FUNCTION_BLOCK FB_PID
VAR_INPUT
	i_bEnablePID		:BOOL	:=FALSE;
	i_rSetpoint			:REAL;				//required input from PLC logic
	i_rActual			:REAL;				//required input from PLC logic
	i_rKp				:REAL;
	i_rKi				:REAL;
	i_rKd				:REAL;
	i_rTdamp			:REAL;
	i_rOutMin			:REAL	:=0;
	i_rOutMax			:REAL	:=100;
	i_rManualOutput		:REAL	:=0;
	i_bEnablePWM		:BOOL	:=FALSE;
	i_iFreqPWM			:INT	:=1000;		//required input from PLC logic
	i_bAutotuneStart	:BOOL	:=FALSE;
	i_rAutotuneSetpoint	:REAL	:=0;
	i_bEnableAlarms		:BOOL;
	i_iHighAlarm		:INT;
	i_iHighWarning		:INT;
	i_iLowWarning		:INT;
	i_iLowAlarm			:INT;
	i_iWarningDelay		:INT;
	i_iAlarmDelay		:INT;
END_VAR
VAR_OUTPUT
	q_rOutputPID		:REAL;				//output for proportional control
	q_bOutputPWM		:BOOL;				//output for on/off control
	q_Difference		:REAL;
	q_AutotuneActive	:BOOL;
	q_AutotuneDone		:BOOL;
	i_sAutotuneTime		:STRING	:='00:00:00';
	q_rAutotuneKp		:REAL	:=0;
	q_rAutotuneKi		:REAL	:=0;
	q_rAutotuneKd		:REAL	:=0;
	q_bError			:BOOL;
	q_bErrorID			:INT	:=0;;
	q_bAlarmHigh		:BOOL;				
	q_bWarningHigh		:BOOL;
	q_bWarningLow		:BOOL;
	q_bAlarmLow			:BOOL;
END_VAR
VAR
	PID_AutoTuner		:FB_PID_AutoTuner;
	PWM_Autotune		:FB_PID_PWM;
	PID_Gain2Time		:FB_PID_Gain2Time;
	ST_PID_Params		:ST_CTRL_PID_PARAMS;
	PID_Control			:FB_CTRL_PID;
	PWM_Control			:FB_PID_PWM;
	M_Active_0			:FB_CTRL_PID;
	
	tonAlarmHigh		:TON;
	tonWarningHigh		:TON;
	tonWarningLow		:TON;
	tonAlarmLow			:TON;
	tonAutotuneTime		:TON;
	
END_VAR
VAR // added by the converter: edge detectors and wires of the graphical bodies
    _w1, _w2, _w3, _w4, _w5 : BOOL;
END_VAR

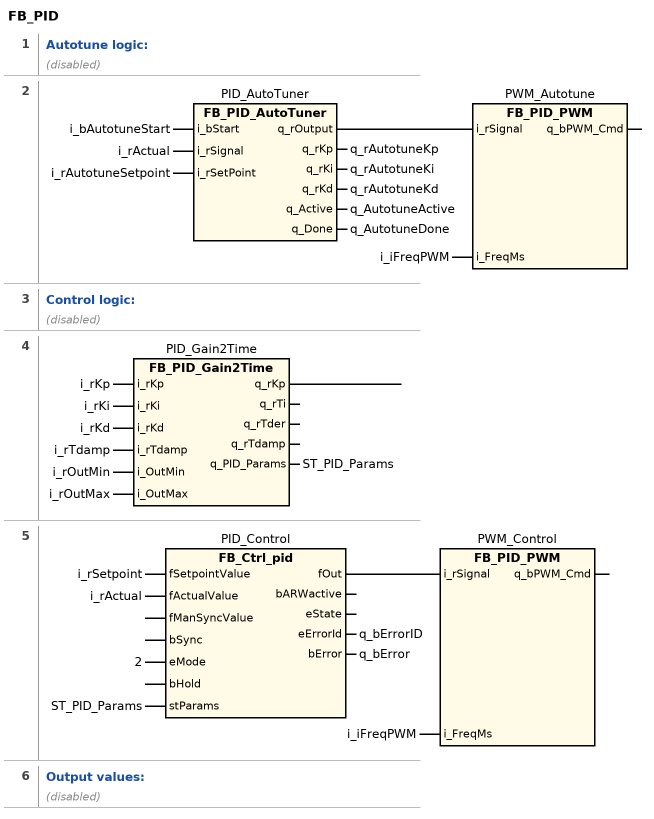
// NETWORK 1 (disabled)
// label: Autotune logic

// NETWORK 2
PID_AutoTuner(
    i_bStart := i_bAutotuneStart,
    i_rSignal := i_rActual,
    i_rSetPoint := i_rAutotuneSetpoint,
    q_rKp => q_rAutotuneKp,
    q_rKi => q_rAutotuneKi,
    q_rKd => q_rAutotuneKd,
    q_Active => q_AutotuneActive,
    q_Done => q_AutotuneDone); // FB_PID_AutoTuner
PWM_Autotune(i_rSignal := PID_AutoTuner.q_rOutput, i_FreqMs := i_iFreqPWM); // FB_PID_PWM

// NETWORK 3 (disabled)
// label: Control logic

// NETWORK 4
PID_Gain2Time(
    i_rKp := i_rKp,
    i_rKi := i_rKi,
    i_rKd := i_rKd,
    i_rTdamp := i_rTdamp,
    i_OutMin := i_rOutMin,
    i_OutMax := i_rOutMax,
    q_PID_Params => ST_PID_Params); // FB_PID_Gain2Time

// NETWORK 5
PID_Control(
    fSetpointValue := i_rSetpoint,
    fActualValue := i_rActual,
    eMode := 2,
    stParams := ST_PID_Params,
    eErrorId => q_bErrorID,
    bError => q_bError); // FB_Ctrl_pid
PWM_Control(i_rSignal := PID_Control.fOut, i_FreqMs := i_iFreqPWM); // FB_PID_PWM

// NETWORK 6 (disabled)
// label: Output values

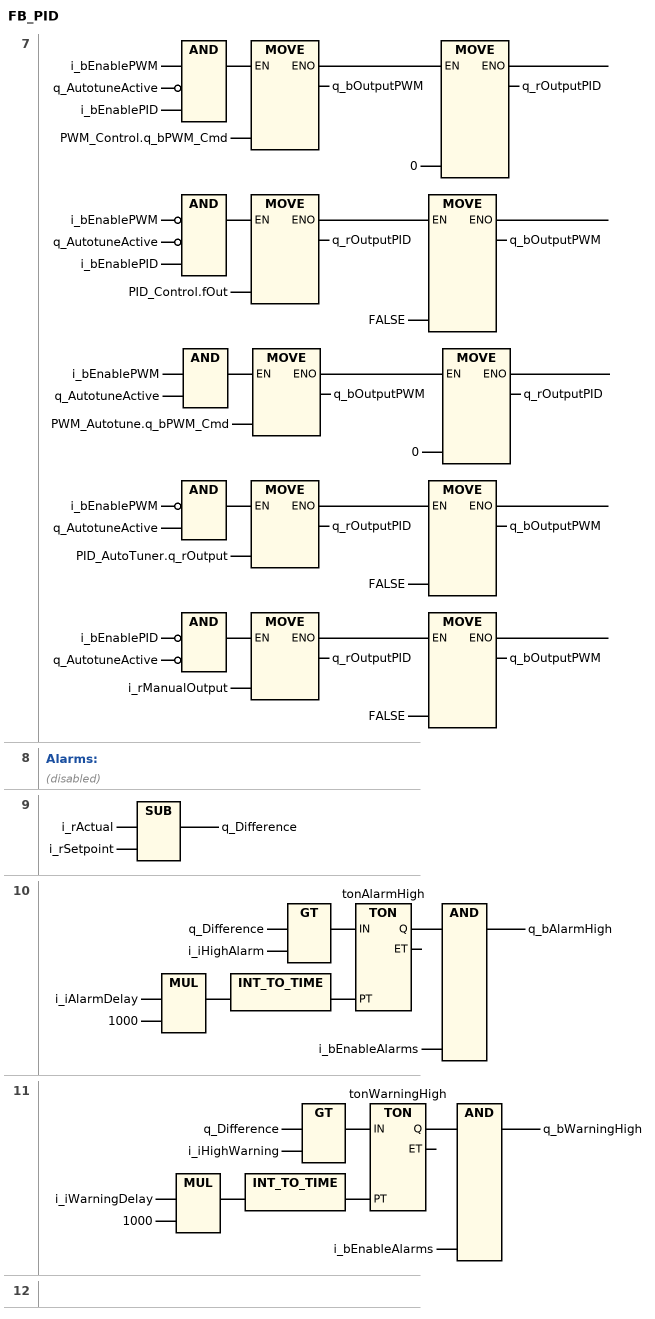
// NETWORK 7
_w1 := i_bEnablePWM AND NOT q_AutotuneActive AND i_bEnablePID;
IF _w1 THEN q_bOutputPWM := PWM_Control.q_bPWM_Cmd; END_IF
IF _w1 THEN q_rOutputPID := 0; END_IF
_w2 := NOT i_bEnablePWM AND NOT q_AutotuneActive AND i_bEnablePID;
IF _w2 THEN q_rOutputPID := PID_Control.fOut; END_IF
IF _w2 THEN q_bOutputPWM := FALSE; END_IF
_w3 := i_bEnablePWM AND q_AutotuneActive;
IF _w3 THEN q_bOutputPWM := PWM_Autotune.q_bPWM_Cmd; END_IF
IF _w3 THEN q_rOutputPID := 0; END_IF
_w4 := NOT i_bEnablePWM AND q_AutotuneActive;
IF _w4 THEN q_rOutputPID := PID_AutoTuner.q_rOutput; END_IF
IF _w4 THEN q_bOutputPWM := FALSE; END_IF
_w5 := NOT i_bEnablePID AND NOT q_AutotuneActive;
IF _w5 THEN q_rOutputPID := i_rManualOutput; END_IF
IF _w5 THEN q_bOutputPWM := FALSE; END_IF

// NETWORK 8 (disabled)
// label: Alarms

// NETWORK 9
q_Difference := i_rActual - i_rSetpoint;

// NETWORK 10
tonAlarmHigh(IN := q_Difference > i_iHighAlarm, PT := INT_TO_TIME(i_iAlarmDelay * 1000)); // TON
q_bAlarmHigh := tonAlarmHigh.Q AND i_bEnableAlarms;

// NETWORK 11
tonWarningHigh(IN := q_Difference > i_iHighWarning, PT := INT_TO_TIME(i_iWarningDelay * 1000)); // TON
q_bWarningHigh := tonWarningHigh.Q AND i_bEnableAlarms;

// NETWORK 12

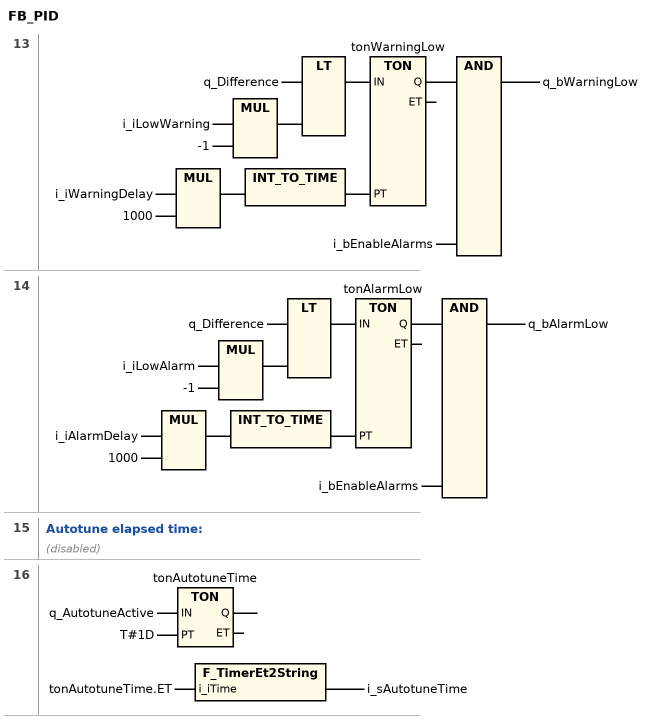
// NETWORK 13
tonWarningLow(IN := q_Difference < i_iLowWarning * -1, PT := INT_TO_TIME(i_iWarningDelay * 1000)); // TON
q_bWarningLow := tonWarningLow.Q AND i_bEnableAlarms;

// NETWORK 14
tonAlarmLow(IN := q_Difference < i_iLowAlarm * -1, PT := INT_TO_TIME(i_iAlarmDelay * 1000)); // TON
q_bAlarmLow := tonAlarmLow.Q AND i_bEnableAlarms;

// NETWORK 15 (disabled)
// label: Autotune elapsed time

// NETWORK 16
tonAutotuneTime(IN := q_AutotuneActive, PT := T#1D); // TON
i_sAutotuneTime := F_TimerEt2String(i_iTime := tonAutotuneTime.ET);

END_FUNCTION_BLOCK

(* stored: Version 1.1.0.1, ProductVersion 3.1.4024.12
   POU FB_PID: Id {a8317d4b-22b8-419a-99b7-52ae7e3313e6}, SpecialFunc None *)
